(* IEC 61131-3 sources: AGA8-92DC_FOR_PLC/CÓDIGOS_AVULSOS, 8 files *)

(* ---- COEF.st ---- *)
VAR_GLOBAL
	K1	: LREAL;
	CNS	: ARRAY [0..57] OF LREAL;
	BI	: ARRAY [0..17] OF LREAL;
END_VAR

(* ---- GRENZDATA.st ---- *)
VAR_GLOBAL
	XN: ARRAY [0..20] OF LREAL :=
	[	50.0,	0.0,	0.0,	0.0,	0.0,	0.0,	0.0,
		 0.0,	0.0,	0.0,	0.0,	0.0,	0.0,	0.0,
		 0.0,	0.0,	0.0,	0.0,	0.0,	0.0,	0.0];

	XH: ARRAY [0..20] OF LREAL :=
	[	100.00,	20.00,	5.000,	1.50,	1.50,	00.5,	00.5,
		000.10,	00.05,	0.050,	0.05,	0.05,	30.0,	50.0,
		000.02,	00.50,	0.015,	0.02,	0.02,	10.0,	03.0];
END_VAR

(* ---- MW.st ---- *)
VAR_GLOBAL
	MWX		: LREAL;
	RGAS	: LREAL;
	TCM		: LREAL;
	DCM		: LREAL;
END_VAR

(* ---- PARAMETERS.st ---- *)
VAR_GLOBAL
	EMW	: ARRAY [0..20] OF LREAL :=
	[	016.0430,	028.0135,	044.0100,	030.0700,
		044.0970,	018.0153,	034.0820,	002.0159,
		028.0100,	031.9988,	058.1230,	058.1230,
		072.1500,	072.1500,	086.1770,	100.2040,
		114.2310,	128.2580,	142.2850,	004.0026,
		039.9480];

	EI	: ARRAY [0..20] OF LREAL :=
	[	151.318300,	099.737780,	241.960600,	244.166700,
		298.118300,	514.015600,	296.355000,	026.957940,
		105.534800,	122.766700,	324.068900,	337.638900,
		365.599900,	370.682300,	402.636293,	427.722630,
		450.325022,	470.840891,	489.558373,	002.610111,
		119.629900];

	KI	: ARRAY [0..20] OF LREAL :=
	[	0.4619255,	0.4479153,	0.4557489,	0.5279209,
		0.5837490,	0.3825868,	0.4618263,	0.3514916,
		0.4533894,	0.4186954,	0.6406937,	0.6341423,
		0.6738577,	0.6798307,	0.7175118,	0.7525189,
		0.7849550,	0.8152731,	0.8437826,	0.3589888,
		0.4216551];

	GI	: ARRAY [0..20] OF LREAL :=
	[	0.000000,	0.027815,	0.189065,	0.079300,	0.141239,
		0.332500,	0.088500,	0.034369,	0.038953,	0.021000,
		0.256692,	0.281835,	0.332267,	0.366911,	0.289731,
		0.337542,	0.383381,	0.427354,	0.469659,	0.000000,
		0.000000];

	QI	: ARRAY [0..20] OF LREAL :=
	[2(0), 0.69, 2(0), 1.06775, 0.633276, 14(0)];

	FI	: ARRAY [0..20] OF LREAL :=
	[7(0), 1, 13(0)];

	SI	: ARRAY [0..20] OF LREAL :=
	[5(0), 1.5822, 0.390, 14(0)];

	WI	: ARRAY [0..20] OF LREAL :=
	[5(0), 1, 15(0)];

	EIJ: ARRAY [0..20, 0..20] OF LREAL :=
	[	1.000000,0.971640,0.960644,1.000000,0.994635,0.708218,0.931484,
		1.170520,0.990126,1.000000,1.019530,0.989844,1.002350,0.999268,
		1.107274,0.880880,0.880973,0.881067,0.881161,1.000000,1.000000,
		1.000000,1.000000,1.022740,0.970120,0.945939,0.746954,0.902271,
		1.086320,1.005710,1.021000,0.946914,0.973384,0.959340,0.945520,
		1.000000,1.000000,1.000000,1.000000,1.000000,1.000000,1.000000,
		1.000000,1.000000,1.000000,0.925053,0.960237,0.849408,0.955052,
		1.281790,1.500000,1.000000,0.906849,0.897362,0.726255,0.859764,
		0.855134,0.831229,0.808310,0.786323,0.765171,1.000000,1.000000,
		1.000000,1.000000,1.000000,1.000000,1.022560,0.693168,0.946871,
		1.164460,1.000000,1.000000,1.000000,1.013060,1.000000,1.005320,
		1.000000,1.000000,1.000000,1.000000,1.000000,1.000000,1.000000,
		1.000000,1.000000,1.000000,1.000000,1.000000,1.000000,1.000000,
		1.034787,1.000000,1.000000,1.000000,1.004900,1.000000,1.000000,
		1.000000,1.000000,1.000000,1.000000,1.000000,1.000000,1.000000,
		1.000000,1.000000,1.000000,1.000000,1.000000,1.000000,1.000000,
		1.000000,1.000000,1.000000,1.000000,1.000000,1.000000,1.000000,
		1.000000,1.000000,1.000000,1.000000,1.000000,1.000000,1.000000,
		1.000000,1.000000,1.000000,1.000000,1.000000,1.000000,1.000000,
		1.000000,1.000000,1.000000,1.000000,1.000000,1.000000,1.000000,
		1.008692,1.010126,1.011501,1.012821,1.014089,1.000000,1.000000,
		1.000000,1.000000,1.000000,1.000000,1.000000,1.000000,1.000000,
		1.000000,1.100000,1.000000,1.300000,1.300000,1.000000,1.000000,
		1.000000,1.000000,1.000000,1.000000,1.000000,1.000000,1.000000,
		1.000000,1.000000,1.000000,1.000000,1.000000,1.000000,1.000000,
		1.000000,1.000000,1.000000,1.000000,1.000000,1.000000,1.000000,
		1.000000,1.000000,1.000000,1.000000,1.000000,1.000000,1.000000,
		1.000000,1.000000,1.000000,1.000000,1.000000,1.000000,1.000000,
		1.000000,1.000000,1.000000,1.000000,1.000000,1.000000,1.000000,
		1.000000,1.000000,1.000000,1.000000,1.000000,1.000000,1.000000,
		1.000000,1.000000,1.000000,1.000000,1.000000,1.000000,1.000000,
		1.000000,1.000000,1.000000,1.000000,1.000000,1.000000,1.000000,
		1.000000,1.000000,1.000000,1.000000,1.000000,1.000000,1.000000,
		1.000000,1.000000,1.000000,1.000000,1.000000,1.000000,1.000000,
		1.000000,1.000000,1.000000,1.000000,1.000000,1.000000,1.000000,
		1.000000,1.000000,1.000000,1.000000,1.000000,1.000000,1.000000,
		1.000000,1.000000,1.000000,1.000000,1.000000,1.000000,1.000000,
		1.000000,1.000000,1.000000,1.000000,1.000000,1.000000,1.000000,
		1.000000,1.000000,1.000000,1.000000,1.000000,1.000000,1.000000,
		1.000000,1.000000,1.000000,1.000000,1.000000,1.000000,1.000000,
		1.000000,1.000000,1.000000,1.000000,1.000000,1.000000,1.000000,
		1.000000,1.000000,1.000000,1.000000,1.000000,1.000000,1.000000,
		1.000000,1.000000,1.000000,1.000000,1.000000,1.000000,1.000000,
		1.000000,1.000000,1.000000,1.000000,1.000000,1.000000,1.000000,
		1.000000,1.000000,1.000000,1.000000,1.000000,1.000000,1.000000,
		1.000000,1.000000,1.000000,1.000000,1.000000,1.000000,1.000000,
		1.000000,1.000000,1.000000,1.000000,1.000000,1.000000,1.000000,
		1.000000,1.000000,1.000000,1.000000,1.000000,1.000000,1.000000,
		1.000000,1.000000,1.000000,1.000000,1.000000,1.000000,1.000000,
		1.000000,1.000000,1.000000,1.000000,1.000000,1.000000,1.000000,
		1.000000,1.000000,1.000000,1.000000,1.000000,1.000000,1.000000,
		1.000000,1.000000,1.000000,1.000000,1.000000,1.000000,1.000000,
		1.000000,1.000000,1.000000,1.000000,1.000000,1.000000,1.000000,
		1.000000,1.000000,1.000000,1.000000,1.000000,1.000000,1.000000,
		1.000000,1.000000,1.000000,1.000000,1.000000,1.000000,1.000000,
		1.000000,1.000000,1.000000,1.000000,1.000000,1.000000,1.000000,
		1.000000,1.000000,1.000000,1.000000,1.000000,1.000000,1.000000,
		1.000000,1.000000,1.000000,1.000000,1.000000,1.000000,1.000000,
		1.000000,1.000000,1.000000,1.000000,1.000000,1.000000,1.000000,
		1.000000,1.000000,1.000000,1.000000,1.000000,1.000000,1.000000,
		1.000000,1.000000,1.000000,1.000000,1.000000,1.000000,1.000000,
		1.000000,1.000000,1.000000,1.000000,1.000000,1.000000,1.000000,
		1.000000,1.000000,1.000000,1.000000,1.000000,1.000000,1.000000];

	UIJ: ARRAY [0..20, 0..20] OF LREAL :=
	[	1.000000,0.886106,0.963827,1.000000,0.990877,1.000000,0.736833,
		1.156390,1.000000,1.000000,1.000000,0.992291,1.000000,1.003670,
		1.302576,1.191904,1.205769,1.219634,1.233498,1.000000,1.000000,
		1.000000,1.000000,0.835058,0.816431,0.915502,1.000000,0.993476,
		0.408838,1.000000,1.000000,1.000000,0.993556,1.000000,1.000000,
		1.000000,1.000000,1.000000,1.000000,1.000000,1.000000,1.000000,
		1.000000,1.000000,1.000000,0.969870,1.000000,1.000000,1.045290,
		1.000000,0.900000,1.000000,1.000000,1.000000,1.000000,1.000000,
		1.066638,1.077634,1.088178,1.098291,1.108021,1.000000,1.000000,
		1.000000,1.000000,1.000000,1.000000,1.065173,1.000000,0.971926,
		1.616660,1.000000,1.000000,1.250000,1.250000,1.250000,1.250000,
		1.000000,1.000000,1.000000,1.000000,1.000000,1.000000,1.000000,
		1.000000,1.000000,1.000000,1.000000,1.000000,1.000000,1.000000,
		1.000000,1.000000,1.000000,1.000000,1.000000,1.000000,1.000000,
		1.000000,1.000000,1.000000,1.000000,1.000000,1.000000,1.000000,
		1.000000,1.000000,1.000000,1.000000,1.000000,1.000000,1.000000,
		1.000000,1.000000,1.000000,1.000000,1.000000,1.000000,1.000000,
		1.000000,1.000000,1.000000,1.000000,1.000000,1.000000,1.000000,
		1.000000,1.000000,1.000000,1.000000,1.000000,1.000000,1.000000,
		1.000000,1.000000,1.000000,1.000000,1.000000,1.000000,1.000000,
		1.028973,1.033754,1.038338,1.042735,1.046966,1.000000,1.000000,
		1.000000,1.000000,1.000000,1.000000,1.000000,1.000000,1.000000,
		1.000000,1.000000,1.000000,1.000000,1.000000,1.000000,1.000000,
		1.000000,1.000000,1.000000,1.000000,1.000000,1.000000,1.000000,
		1.000000,1.000000,1.000000,1.000000,1.000000,1.000000,1.000000,
		1.000000,1.000000,1.000000,1.000000,1.000000,1.000000,1.000000,
		1.000000,1.000000,1.000000,1.000000,1.000000,1.000000,1.000000,
		1.000000,1.000000,1.000000,1.000000,1.000000,1.000000,1.000000,
		1.000000,1.000000,1.000000,1.000000,1.000000,1.000000,1.000000,
		1.000000,1.000000,1.000000,1.000000,1.000000,1.000000,1.000000,
 		1.000000,1.000000,1.000000,1.000000,1.000000,1.000000,1.000000,
		1.000000,1.000000,1.000000,1.000000,1.000000,1.000000,1.000000,
		1.000000,1.000000,1.000000,1.000000,1.000000,1.000000,1.000000,
 		1.000000,1.000000,1.000000,1.000000,1.000000,1.000000,1.000000,
		1.000000,1.000000,1.000000,1.000000,1.000000,1.000000,1.000000,
		1.000000,1.000000,1.000000,1.000000,1.000000,1.000000,1.000000,
		1.000000,1.000000,1.000000,1.000000,1.000000,1.000000,1.000000,
		1.000000,1.000000,1.000000,1.000000,1.000000,1.000000,1.000000,
		1.000000,1.000000,1.000000,1.000000,1.000000,1.000000,1.000000,
		1.000000,1.000000,1.000000,1.000000,1.000000,1.000000,1.000000,
		1.000000,1.000000,1.000000,1.000000,1.000000,1.000000,1.000000,
		1.000000,1.000000,1.000000,1.000000,1.000000,1.000000,1.000000,
		1.000000,1.000000,1.000000,1.000000,1.000000,1.000000,1.000000,
		1.000000,1.000000,1.000000,1.000000,1.000000,1.000000,1.000000,
		1.000000,1.000000,1.000000,1.000000,1.000000,1.000000,1.000000,
		1.000000,1.000000,1.000000,1.000000,1.000000,1.000000,1.000000,
		1.000000,1.000000,1.000000,1.000000,1.000000,1.000000,1.000000,
		1.000000,1.000000,1.000000,1.000000,1.000000,1.000000,1.000000,
		1.000000,1.000000,1.000000,1.000000,1.000000,1.000000,1.000000,
		1.000000,1.000000,1.000000,1.000000,1.000000,1.000000,1.000000,
		1.000000,1.000000,1.000000,1.000000,1.000000,1.000000,1.000000,
		1.000000,1.000000,1.000000,1.000000,1.000000,1.000000,1.000000,
		1.000000,1.000000,1.000000,1.000000,1.000000,1.000000,1.000000,
		1.000000,1.000000,1.000000,1.000000,1.000000,1.000000,1.000000,
		1.000000,1.000000,1.000000,1.000000,1.000000,1.000000,1.000000,
		1.000000,1.000000,1.000000,1.000000,1.000000,1.000000,1.000000,
		1.000000,1.000000,1.000000,1.000000,1.000000,1.000000,1.000000,
		1.000000,1.000000,1.000000,1.000000,1.000000,1.000000,1.000000,
		1.000000,1.000000,1.000000,1.000000,1.000000,1.000000,1.000000,
		1.000000,1.000000,1.000000,1.000000,1.000000,1.000000,1.000000,
		1.000000,1.000000,1.000000,1.000000,1.000000,1.000000,1.000000,
		1.000000,1.000000,1.000000,1.000000,1.000000,1.000000,1.000000,
		1.000000,1.000000,1.000000,1.000000,1.000000,1.000000,1.000000];

	KIJ: ARRAY [0..20, 0..20] OF LREAL :=
	[	1.000000,1.003630,0.995933,1.000000,1.007619,1.000000,1.000080,
		1.023260,1.000000,1.000000,1.000000,0.997596,1.000000,1.002529,
		0.982962,0.983565,0.982707,0.981849,0.980991,1.000000,1.000000,
		1.000000,1.000000,0.982361,1.007960,1.000000,1.000000,0.942596,
		1.032270,1.000000,1.000000,1.000000,1.000000,1.000000,1.000000,
		1.000000,1.000000,1.000000,1.000000,1.000000,1.000000,1.000000,
		1.000000,1.000000,1.000000,1.008510,1.000000,1.000000,1.007790,
		1.000000,1.000000,1.000000,1.000000,1.000000,1.000000,1.000000,
		0.910183,0.895362,0.881152,0.867520,0.854406,1.000000,1.000000,
		1.000000,1.000000,1.000000,1.000000,0.986893,1.000000,0.999969,
		1.020340,1.000000,1.000000,1.000000,1.000000,1.000000,1.000000,
		1.000000,1.000000,1.000000,1.000000,1.000000,1.000000,1.000000,
		1.000000,1.000000,1.000000,1.000000,1.000000,1.000000,1.000000,
		1.000000,1.000000,1.000000,1.000000,1.000000,1.000000,1.000000,
		1.000000,1.000000,1.000000,1.000000,1.000000,1.000000,1.000000,
		1.000000,1.000000,1.000000,1.000000,1.000000,1.000000,1.000000,
		1.000000,1.000000,1.000000,1.000000,1.000000,1.000000,1.000000,
		1.000000,1.000000,1.000000,1.000000,1.000000,1.000000,1.000000,
		1.000000,1.000000,1.000000,1.000000,1.000000,1.000000,1.000000,
		1.000000,1.000000,1.000000,1.000000,1.000000,1.000000,1.000000,
		0.968130,0.962870,0.957828,0.952441,0.948338,1.000000,1.000000,
		1.000000,1.000000,1.000000,1.000000,1.000000,1.000000,1.000000,
		1.000000,1.000000,1.000000,1.000000,1.000000,1.000000,1.000000,
		1.000000,1.000000,1.000000,1.000000,1.000000,1.000000,1.000000,
		1.000000,1.000000,1.000000,1.000000,1.000000,1.000000,1.000000,
		1.000000,1.000000,1.000000,1.000000,1.000000,1.000000,1.000000,
		1.000000,1.000000,1.000000,1.000000,1.000000,1.000000,1.000000,
		1.000000,1.000000,1.000000,1.000000,1.000000,1.000000,1.000000,
		1.000000,1.000000,1.000000,1.000000,1.000000,1.000000,1.000000,
		1.000000,1.000000,1.000000,1.000000,1.000000,1.000000,1.000000,
		1.000000,1.000000,1.000000,1.000000,1.000000,1.000000,1.000000,
		1.000000,1.000000,1.000000,1.000000,1.000000,1.000000,1.000000,
		1.000000,1.000000,1.000000,1.000000,1.000000,1.000000,1.000000,
		1.000000,1.000000,1.000000,1.000000,1.000000,1.000000,1.000000,
		1.000000,1.000000,1.000000,1.000000,1.000000,1.000000,1.000000,
		1.000000,1.000000,1.000000,1.000000,1.000000,1.000000,1.000000,
		1.000000,1.000000,1.000000,1.000000,1.000000,1.000000,1.000000,
		1.000000,1.000000,1.000000,1.000000,1.000000,1.000000,1.000000,
		1.000000,1.000000,1.000000,1.000000,1.000000,1.000000,1.000000,
		1.000000,1.000000,1.000000,1.000000,1.000000,1.000000,1.000000,
		1.000000,1.000000,1.000000,1.000000,1.000000,1.000000,1.000000,
		1.000000,1.000000,1.000000,1.000000,1.000000,1.000000,1.000000,
		1.000000,1.000000,1.000000,1.000000,1.000000,1.000000,1.000000,
		1.000000,1.000000,1.000000,1.000000,1.000000,1.000000,1.000000,
		1.000000,1.000000,1.000000,1.000000,1.000000,1.000000,1.000000,
		1.000000,1.000000,1.000000,1.000000,1.000000,1.000000,1.000000,
		1.000000,1.000000,1.000000,1.000000,1.000000,1.000000,1.000000,
		1.000000,1.000000,1.000000,1.000000,1.000000,1.000000,1.000000,
		1.000000,1.000000,1.000000,1.000000,1.000000,1.000000,1.000000,
		1.000000,1.000000,1.000000,1.000000,1.000000,1.000000,1.000000,
		1.000000,1.000000,1.000000,1.000000,1.000000,1.000000,1.000000,
		1.000000,1.000000,1.000000,1.000000,1.000000,1.000000,1.000000,
		1.000000,1.000000,1.000000,1.000000,1.000000,1.000000,1.000000,
		1.000000,1.000000,1.000000,1.000000,1.000000,1.000000,1.000000,
		1.000000,1.000000,1.000000,1.000000,1.000000,1.000000,1.000000,
		1.000000,1.000000,1.000000,1.000000,1.000000,1.000000,1.000000,
		1.000000,1.000000,1.000000,1.000000,1.000000,1.000000,1.000000,
		1.000000,1.000000,1.000000,1.000000,1.000000,1.000000,1.000000,
		1.000000,1.000000,1.000000,1.000000,1.000000,1.000000,1.000000,
		1.000000,1.000000,1.000000,1.000000,1.000000,1.000000,1.000000,
		1.000000,1.000000,1.000000,1.000000,1.000000,1.000000,1.000000,
		1.000000,1.000000,1.000000,1.000000,1.000000,1.000000,1.000000,
		1.000000,1.000000,1.000000,1.000000,1.000000,1.000000,1.000000];

	GIJ: ARRAY [0..20, 0..20] OF LREAL :=
	[	1.000000,1.000000,0.807653,1.000000,1.000000,1.000000,1.000000,
		1.957310,1.000000,1.000000,1.000000,1.000000,1.000000,1.000000,
		1.000000,1.000000,1.000000,1.000000,1.000000,1.000000,1.000000,
		1.000000,1.000000,0.982746,1.000000,1.000000,1.000000,1.000000,
		1.000000,1.000000,1.000000,1.000000,1.000000,1.000000,1.000000,
		1.000000,1.000000,1.000000,1.000000,1.000000,1.000000,1.000000,
		1.000000,1.000000,1.000000,0.370296,1.000000,1.673090,1.000000,
		1.000000,1.000000,1.000000,1.000000,1.000000,1.000000,1.000000,
		1.000000,1.000000,1.000000,1.000000,1.000000,1.000000,1.000000,
		1.000000,1.000000,1.000000,1.000000,1.000000,1.000000,1.000000,
		1.000000,1.000000,1.000000,1.000000,1.000000,1.000000,1.000000,
		1.000000,1.000000,1.000000,1.000000,1.000000,1.000000,1.000000,
		1.000000,1.000000,1.000000,1.000000,1.000000,1.000000,1.000000,
		1.000000,1.000000,1.000000,1.000000,1.000000,1.000000,1.000000,
		1.000000,1.000000,1.000000,1.000000,1.000000,1.000000,1.000000,
		1.000000,1.000000,1.000000,1.000000,1.000000,1.000000,1.000000,
		1.000000,1.000000,1.000000,1.000000,1.000000,1.000000,1.000000,
		1.000000,1.000000,1.000000,1.000000,1.000000,1.000000,1.000000,
		1.000000,1.000000,1.000000,1.000000,1.000000,1.000000,1.000000,
		1.000000,1.000000,1.000000,1.000000,1.000000,1.000000,1.000000,
		1.000000,1.000000,1.000000,1.000000,1.000000,1.000000,1.000000,
		1.000000,1.000000,1.000000,1.000000,1.000000,1.000000,1.000000,
		1.000000,1.000000,1.000000,1.000000,1.000000,1.000000,1.000000,
		1.000000,1.000000,1.000000,1.000000,1.000000,1.000000,1.000000,
		1.000000,1.000000,1.000000,1.000000,1.000000,1.000000,1.000000,
		1.000000,1.000000,1.000000,1.000000,1.000000,1.000000,1.000000,
		1.000000,1.000000,1.000000,1.000000,1.000000,1.000000,1.000000,
		1.000000,1.000000,1.000000,1.000000,1.000000,1.000000,1.000000,
		1.000000,1.000000,1.000000,1.000000,1.000000,1.000000,1.000000,
		1.000000,1.000000,1.000000,1.000000,1.000000,1.000000,1.000000,
		1.000000,1.000000,1.000000,1.000000,1.000000,1.000000,1.000000,
		1.000000,1.000000,1.000000,1.000000,1.000000,1.000000,1.000000,
		1.000000,1.000000,1.000000,1.000000,1.000000,1.000000,1.000000,
		1.000000,1.000000,1.000000,1.000000,1.000000,1.000000,1.000000,
		1.000000,1.000000,1.000000,1.000000,1.000000,1.000000,1.000000,
		1.000000,1.000000,1.000000,1.000000,1.000000,1.000000,1.000000,
		1.000000,1.000000,1.000000,1.000000,1.000000,1.000000,1.000000,
		1.000000,1.000000,1.000000,1.000000,1.000000,1.000000,1.000000,
		1.000000,1.000000,1.000000,1.000000,1.000000,1.000000,1.000000,
		1.000000,1.000000,1.000000,1.000000,1.000000,1.000000,1.000000,
		1.000000,1.000000,1.000000,1.000000,1.000000,1.000000,1.000000,
		1.000000,1.000000,1.000000,1.000000,1.000000,1.000000,1.000000,
		1.000000,1.000000,1.000000,1.000000,1.000000,1.000000,1.000000,
		1.000000,1.000000,1.000000,1.000000,1.000000,1.000000,1.000000,
		1.000000,1.000000,1.000000,1.000000,1.000000,1.000000,1.000000,
		1.000000,1.000000,1.000000,1.000000,1.000000,1.000000,1.000000,
		1.000000,1.000000,1.000000,1.000000,1.000000,1.000000,1.000000,
		1.000000,1.000000,1.000000,1.000000,1.000000,1.000000,1.000000,
		1.000000,1.000000,1.000000,1.000000,1.000000,1.000000,1.000000,
		1.000000,1.000000,1.000000,1.000000,1.000000,1.000000,1.000000,
		1.000000,1.000000,1.000000,1.000000,1.000000,1.000000,1.000000,
		1.000000,1.000000,1.000000,1.000000,1.000000,1.000000,1.000000,
		1.000000,1.000000,1.000000,1.000000,1.000000,1.000000,1.000000,
		1.000000,1.000000,1.000000,1.000000,1.000000,1.000000,1.000000,
		1.000000,1.000000,1.000000,1.000000,1.000000,1.000000,1.000000,
		1.000000,1.000000,1.000000,1.000000,1.000000,1.000000,1.000000,
		1.000000,1.000000,1.000000,1.000000,1.000000,1.000000,1.000000,
		1.000000,1.000000,1.000000,1.000000,1.000000,1.000000,1.000000,
		1.000000,1.000000,1.000000,1.000000,1.000000,1.000000,1.000000,
		1.000000,1.000000,1.000000,1.000000,1.000000,1.000000,1.000000,
		1.000000,1.000000,1.000000,1.000000,1.000000,1.000000,1.000000,
		1.000000,1.000000,1.000000,1.000000,1.000000,1.000000,1.000000,
		1.000000,1.000000,1.000000,1.000000,1.000000,1.000000,1.000000];
END_VAR

(* ---- DCAGA.st ---- *)
FUNCTION DCAGA : BOOL
VAR_INPUT
	XJ : ARRAY [0..20] OF LREAL;
END_VAR

VAR
	I		: INT						;
	J		: INT						;
	N		: INT						;
	SUM		: LREAL						;
	XI		: ARRAY [0..20] OF LREAL	;
	U1		: LREAL						;
	G1		: LREAL						;
	Q1		: LREAL						;
	F1		: LREAL						;
	E1		: LREAL						;
	XIJ		: LREAL						;
	EIJ0	: LREAL						;
	GIJ0	: LREAL						;
	BN		: LREAL						;
END_VAR

FOR I:=0 TO 20 DO
	XI[I] := XJ[I];
END_FOR

SUM		:= 0;
MW.MWX	:= 0;

FOR I:=0 TO 20 DO
	SUM := SUM + XI[I];
END_FOR

FOR I:=0 TO 20 DO
	XI[I] := XI[I]/SUM;
END_FOR

MW.RGAS	:= 8.31451E-3;
MW.MWX	:= 0;

FOR I:=0 TO 21 DO
	MW.MWX := MW.MWX + XI[I]* PARAMETERS.EMW[I];
END_FOR

FOR N:=0 TO 17 DO
	COEF.BI[N] := 0;
END_FOR

COEF.K1	:= 0;
U1		:= 0;
G1		:= 0;
Q1		:= 0;
F1		:= 0;
E1		:= 0;

FOR I:=0 TO 20 DO
	COEF.K1 := COEF.K1 + XI[I]*EXPT(PARAMETERS.KI[I],2.5);
 	U1 := U1 + XI[I]*EXPT(PARAMETERS.EI[I],2.5);
 	G1 := G1 + XI[I]*PARAMETERS.GI[I];
 	Q1 := Q1 + XI[I]*PARAMETERS.QI[I];
 	F1 := F1 + XI[I]*XI[I]*PARAMETERS.SI[I];
 	E1 := E1 + XI[I]*PARAMETERS.EI[I];
END_FOR

MW.TCM	:= 1.261*E1;
MW.DCM	:= EXPT(COEF.K1,-1.2);
COEF.K1	:= COEF.K1*COEF.K1;
U1		:= U1*U1;

 FOR I:=0 TO 7 DO
	FOR J:=I+1 TO 18 DO
		XIJ := XI[I]*XI[J];
 			IF (XIJ <> 0) THEN
				COEF.K1 := COEF.K1 + 2.0 * XIJ * (EXPT(PARAMETERS.KIJ[I,J],5)-1) * EXPT((PARAMETERS.KI[I]*PARAMETERS.KI[J]),2.5);
				U1 		:= U1 + 2.0 * XIJ * (EXPT(PARAMETERS.UIJ[I,J],5)-1) * EXPT((PARAMETERS.EI[I]*PARAMETERS.EI[J]),2.5);
				G1 		:= G1 + XIJ * (PARAMETERS.GIJ[I,J] - 1) * (PARAMETERS.GI[I] + PARAMETERS.GI[J]);
 			END_IF
 	END_FOR
END_FOR

FOR I:=0 TO 20 DO
	FOR J:=I TO 20 DO
		XIJ := XI[I]*XI[J];
 		IF (XIJ <> 0) THEN
			IF (I <> J) THEN
				XIJ := 2.0*XIJ;
			END_IF
			EIJ0 := PARAMETERS.EIJ[I,J] * SQRT(PARAMETERS.EI[I]*PARAMETERS.EI[J]);
			GIJ0 := PARAMETERS.GIJ[I,J] * (PARAMETERS.GI[I] + PARAMETERS.GI[J])/2.0;
 			FOR N:=0 TO 17 DO
	 			BN		:= EXPT((GIJ0 + 1.0 - CONSTANTS.G[N]),CONSTANTS.G[N])
						* EXPT((PARAMETERS.QI[I]*PARAMETERS.QI[J] + 1.0 - CONSTANTS.Q[N]),CONSTANTS.Q[N])
 						* EXPT((SQRT(PARAMETERS.SI[I]*PARAMETERS.SI[J]) + 1.0 - CONSTANTS.F[N]),CONSTANTS.F[N])
						* EXPT((PARAMETERS.SI[I]*PARAMETERS.SI[J] + 1.0 - CONSTANTS.S1[N]),CONSTANTS.S1[N])
						* EXPT((PARAMETERS.WI[I]*PARAMETERS.WI[J] + 1.0 - CONSTANTS.W[N]),CONSTANTS.W[N]);
				COEF.BI[N]	:= COEF.BI[N]+CONSTANTS.A[N]*XIJ*EXPT(EIJ0,CONSTANTS.U[N])*EXPT((PARAMETERS.KI[I]*PARAMETERS.KI[J]),1.50)*BN;
			END_FOR
 		END_IF
	END_FOR
END_FOR

COEF.K1 := EXPT(COEF.K1,0.2);
U1 		:= EXPT(U1,0.2);

FOR N:=12 TO 57 DO
	COEF.CNS[N]	:= EXPT((G1 + 1.0 - CONSTANTS.G[N]),CONSTANTS.G[N])
				* EXPT((EXPT(Q1,2) + 1.0 - CONSTANTS.Q[N]),CONSTANTS.Q[N])
				* EXPT((F1 + 1.0 - CONSTANTS.F[N]),CONSTANTS.F[N]) * CONSTANTS.A[N]*EXPT(U1,CONSTANTS.U[N]);
END_FOR

(* ---- DZOFPT.st ---- *)
FUNCTION  DZOFPT : LREAL
VAR_INPUT
	EP		: DWORD;
	ET		: DWORD;
	ED		: DWORD;
	EZ		: DWORD;
	EBmix	: DWORD;
END_VAR
VAR
	P		: POINTER TO LREAL;
	T		: POINTER TO LREAL;
	D		: POINTER TO LREAL;
	Z		: POINTER TO LREAL;
	Bmix	: POINTER TO LREAL;
	X1		: LREAL;
	X2		: LREAL;
	X3		: LREAL;
	F		: LREAL;
	F1		: LREAL;
	F2		: LREAL;
	F3		: LREAL;
	TOL		: LREAL;
	I		: INT;
END_VAR

P		:= EP;
T		:= ET;
D		:= ED;
Z		:= EZ;
Bmix	:= EBmix;

TOL	:= 0.5E-9;
X1	:= 0.0000010;
X2	:= 40.0;
D^	:= 0;

PZOFDT(ED:=ADR(X1), ET:=T, EP:=ADR(F1), EZ:=Z, EBmix:=Bmix);
PZOFDT(ED:=ADR(X2), ET:=T, EP:=ADR(F2), EZ:=Z, EBmix:=Bmix);

F1 := F1 - P^;
F2 := F2 - P^;

IF ((F1*F2)>=0) THEN
	RETURN;
END_IF

FOR I := 0 TO 49 DO
	X3	:= X1 - F1*(X2 - X1)/(F2 - F1);
 	PZOFDT(ED:=ADR(X3), ET:=T, EP:=ADR(F3), EZ:=Z, EBmix:=Bmix);
 	F3	:= F3 - P^;
	D^	:= X1*F2*F3/((F1 - F2)*(F1 - F3))
		+  X2*F1*F3/((F2 - F1)*(F2 - F3))
		+  X3*F1*F2/((F3 - F1)*(F3 - F2));

 	IF ((D^ - X1)*(D^ - X2)>= 0) THEN
		D^ := (X1 + X2)/2.0;
	END_IF

 	PZOFDT(ED:=ADR(D), ET:=T, EP:=ADR(F), EZ:=Z, EBmix:=Bmix);
	F := F - P^;

	IF (ABS(F)<=TOL) THEN
		RETURN;
	END_IF

	IF (ABS(F3)< ABS(F)) AND ((F*F3)>0) THEN
 		IF ((F3*F1)>0) THEN
 			X1 := X3;
 			F1 := F3;
 		ELSE
 			X2 := X3;
 			F2 := F3;
 		END_IF
 	ELSE
 		IF ((F*F3)>0) THEN
 			X1 := D^;
 			F1 := F;
 			X2 := X3;
 			F2 := F3;
 		ELSIF ((F3*F1)>0) THEN
			 X1 := D^;
 			 F1 := F;
 		ELSE
 			 X2 := D^;
 			 F2 := F;
 		END_IF
 	END_IF
 END_FOR

(* ---- PZOFDT.st ---- *)
FUNCTION PZOFDT : LREAL
VAR_INPUT
	ED		: DWORD;
	ET		: DWORD;
	EP		: DWORD;
	EZ		: DWORD;
	EBmix	: DWORD;
END_VAR

VAR
	D		: POINTER TO LREAL	;
	T		: POINTER TO LREAL	;
	P		: POINTER TO LREAL	;
	Z		: POINTER TO LREAL	;
	Bmix	: POINTER TO LREAL	;
	N		: INT				;
  	DR		: LREAL				;
END_VAR

P		:= EP;
T		:= ET;
D		:= ED;
Z		:= EZ;
Bmix	:= EBmix;
DR		:= D^*EXPT(COEF.K1,3);
Bmix^	:= 0;

FOR N:=0 TO 17 DO
	Bmix^ := Bmix^ + COEF.BI[N]/EXPT(T^,CONSTANTS.U[N]);
END_FOR

Z^ := 1.0 + Bmix^ * D^;

FOR N:=12 TO 17 DO
	Z^ := Z^ - DR * COEF.CNS[N]/EXPT(T^,CONSTANTS.U[N]);
END_FOR

FOR N:=12 TO 57 DO
	Z^	:= Z^
		+ COEF.CNS[N]/EXPT(T^,CONSTANTS.U[N])
		*(CONSTANTS.B[N] - CONSTANTS.C[N]*CONSTANTS.K[N]*EXPT(DR,CONSTANTS.K[N]))
		* EXPT(DR,CONSTANTS.B[N])
		* EXP(-CONSTANTS.C[N]*EXPT(DR,CONSTANTS.K[N]));
END_FOR

P^		:= D^ * MW.RGAS * T^ * Z^;
PZOFDT	:= Z^;

(* ---- AGA8_92DC_TESTE.st ---- *)
PROGRAM AGA8_92DC_TESTE
VAR
	Gas_Teste: ARRAY [0..20] OF LREAL :=
	[	0.9650, 0.0030, 0.0060, 0.0180, 0.0045, 0.0000, 0.0000,
		0.0000, 0.0000, 0.0000, 0.0010, 0.0010, 0.0005, 0.0003,
		0.0007, 0.0000, 0.0000, 0.0000, 0.0000, 0.0000, 0.0000];

	T_Teste	: LREAL := 56.85;
	P_Teste	: LREAL := 60.00;

	T_Gas	: LREAL := 0;
	P_Gas	: LREAL := 0;
	Z_Gas	: LREAL := 0;

	Bmix	: LREAL	:=	0;
	D		: LREAL	:=	0;
	P		: LREAL	:=	0;
	T		: LREAL	:= 	0;
	Z		: LREAL	:=	0;
END_VAR

Bmix	:= 0;
D		:= 0;
Z		:= 0;

P		:= P_Teste / 010.00;
P_Gas	:= P_Teste / 010.00;
T		:= T_Teste + 273.15;
T_Gas	:= T_Teste + 273.15;

DCAGA	(XJ:= Gas_Teste);
DZOFPT	(ADR(P), ADR(T), ADR(D), ADR(Z), ADR(Bmix));

Z_Gas:=	PZOFDT(ADR(D), ADR(T), ADR(P), ADR(Z), ADR(Bmix));
